INTERFACE I_CalcImageDistance EXTENDS I_Fallible


METHOD Calculate : LREAL
VAR_INPUT
    fFocalLength : LREAL;
    fSourceDistance : LREAL;
END_VAR
END_METHOD

END_INTERFACE

(* stored: Version 1.1.0.1
   Itf I_CalcImageDistance: Id {9de12eff-520d-467e-99ab-024e0bc23921}
   Method Calculate: Id {73a9a5ee-8e75-47d0-bbff-d8be94099a30} *)
